(* PLC project Rasi_feeds_batching.project, Automation Builder 2.7 - Basic Automation Builder 2.7 *)
(* stored: creationDateTime 2026-08-29T13:26:29.0230133, modificationDateTime 2026-08-29T13:22:02.2412807 *)

CONFIGURATION Application
  RESOURCE Application ON PLC
    TASK Task(INTERVAL := T#10ms, PRIORITY := 14);
    PROGRAM batching13 WITH Task : batching13;
  END_RESOURCE
END_CONFIGURATION
